TYPE CMD_Trolley :
STRUCT
	cmd			: eTcaTrolleyCmd;
	nId			: INT;
END_STRUCT
END_TYPE

(* stored: Version 1.1.0.1
   DUT CMD_Trolley: Id {9e5a0e07-0fe0-4374-914e-d3473a457467} *)
